// TIA Portal V17 export
// export: Created 2024-09-15T12:30:25.6219238Z, ExportSetting WithDefaults, DisplayName Totally Integrated Automation Portal, DisplayVersion V17, DisplayName TIA Portal Openness, DisplayVersion V17, DisplayName TIA Portal Version Control Interface, DisplayVersion V17, DisplayName STEP 7 Professional, DisplayVersion V17, DisplayName STEP 7 Safety, DisplayVersion V17, DisplayName WinCC Professional, DisplayVersion V17
TYPE "typ_State_Client"
// stored: IsFailsafeCompliant false
   STRUCT
      ldt_ts : LDT;
      x_sensor_oven : Bool;
      s_station : String;
      i_code : Int;
      s_description : String;
      x_active : Bool;
      s_target : String;
      x_error : Bool;
      s_errorMessage : String := 'No error';
      Workpiece : "typ_Workpiece";
   END_STRUCT;
END_TYPE
